INTERFACE I_HttpResponse EXTENDS I_Disposable

PROPERTY PUBLIC Json : I_JsonPath
GET
END_GET
END_PROPERTY

PROPERTY PUBLIC ResponseCode : udint
GET
END_GET
END_PROPERTY

END_INTERFACE

(* stored: Version 1.1.0.1, ProductVersion 3.1.4024.12
   Itf I_HttpResponse: Id {51a83b02-023a-06f8-10aa-8a229dd628e0}
   Property Json: Id {9e9bd29b-0414-0bc9-23da-ad86ed7a6dec}
   Get Get: Id {64ba1d36-d431-04d5-0e00-567adbfc79cc}
   Property ResponseCode: Id {2b6ab977-22c9-0a88-2858-067343e938ff}
   Get Get: Id {c4ccf432-1efa-0875-04f7-adb15e39bfc3} *)
